FUNCTION_BLOCK FB_BaseComplexElement_HMI EXTENDS FB_BaseExecutiveElement_HMI IMPLEMENTS ITF_BaseComplexElement_HMI
VAR
	itfBaseComplexElementConnector		: ITF_BaseComplexElement_HMI_Connector;
	refstBaseComplexElementDataHMI		: REFERENCE TO ST_BaseComplexElement_HMI;
END_VAR

END_FUNCTION_BLOCK

(* stored: Version 1.1.0.1
   POU FB_BaseComplexElement_HMI: Id {3f198324-9925-0fb3-39d4-b6620e2a327f}, SpecialFunc None *)
